{attribute 'qualified_only'}
VAR_GLOBAL
    // WPF与PLC的通信握手、心跳及看门狗反馈。
    Comm : ST_HmiCommunication;
END_VAR

(* stored: Version 1.1.0.1, ProductVersion 3.1.4026.18
   GVL GVL_HMI: Id {65f78e28-9d20-414e-8a89-341c4c061362} *)
